{attribute 'qualified_only'}
VAR_GLOBAL 
	A1 AT %I* : ARRAY[0..7] OF BOOL;
	A2 AT %Q* : ARRAY[0..7] OF BOOL;
END_VAR

(* stored: Version 1.1.0.1, ProductVersion 3.1.4024.5
   GVL IO: Id {fa9f344e-05bf-4ebb-872e-4e733cbd3fe1} *)
